{attribute 'GeneratedUsingTerminal: KL3064'}
{attribute addProperty BoxType "KL3064"}
{attribute addProperty Id "Channel_1AT %Q*Channel_6576A6810Channel_2AT %Q*Channel_6576A6810Channel_3AT %Q*Channel_6576A6810Channel_4AT %Q*Channel_6576A6810"}
{attribute addProperty CRC "2346945397"}
{attribute addProperty Size "0"}
TYPE KL3064_8BE38B75 :
STRUCT
	{attribute addProperty Name "Channel_1"}
	Channel_1 : Channel_6576A681;
	{attribute addProperty Name "Channel_2"}
	Channel_2 : Channel_6576A681;
	{attribute addProperty Name "Channel_3"}
	Channel_3 : Channel_6576A681;
	{attribute addProperty Name "Channel_4"}
	Channel_4 : Channel_6576A681;
END_STRUCT
END_TYPE
